FUNCTION_BLOCK POU_MainFunc
VAR_INPUT
END_VAR
VAR_OUTPUT
END_VAR
VAR
	go: BOOL; //local variable to start the program and modes
	TON_0: TON;
	timepass: TIME;
	TimerAmount: TIME:= T#340MS; //this is a specific value type, time of 340ms
	timer2: BOOL;
	Timer1: BOOL;
	TON_1: TON;
	InManual: BOOL;
	Motor: MC_Power;
	onMotor: BOOL;
	Motormove: MC_MoveVelocity;
END_VAR

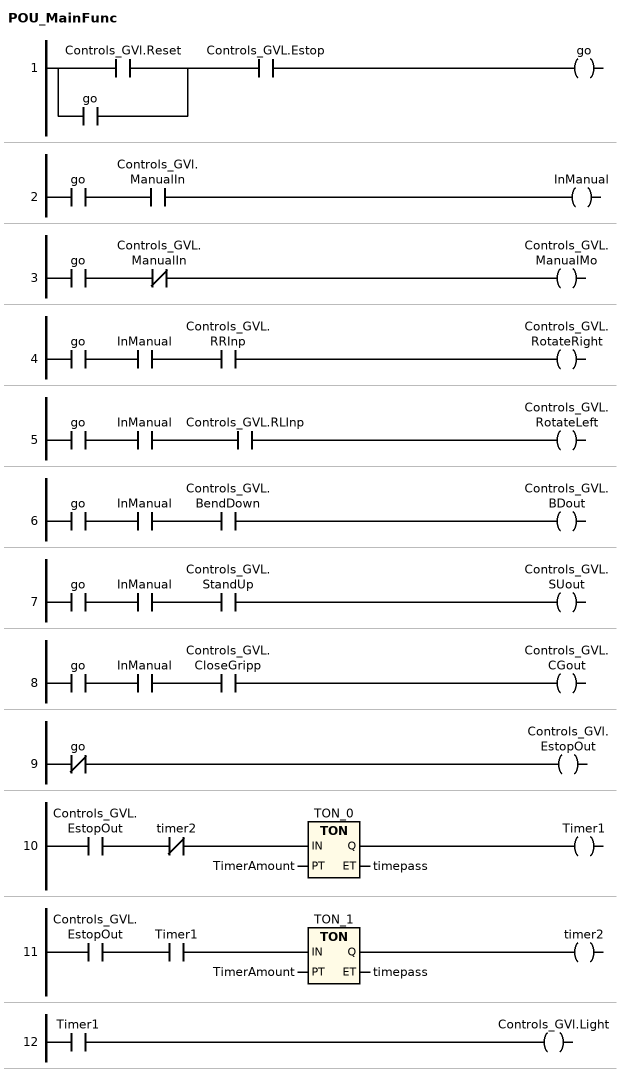
// NETWORK 1
go := (Controls_GVl.Reset OR go) AND Controls_GVL.Estop;

// NETWORK 2
InManual := go AND Controls_GVl.ManualIn;

// NETWORK 3
Controls_GVL.ManualMo := go AND NOT Controls_GVL.ManualIn;

// NETWORK 4
Controls_GVL.RotateRight := go AND InManual AND Controls_GVL.RRInp;

// NETWORK 5
Controls_GVL.RotateLeft := go AND InManual AND Controls_GVL.RLInp;

// NETWORK 6
Controls_GVL.BDout := go AND InManual AND Controls_GVL.BendDown;

// NETWORK 7
Controls_GVL.SUout := go AND InManual AND Controls_GVL.StandUp;

// NETWORK 8
Controls_GVL.CGout := go AND InManual AND Controls_GVL.CloseGripp;

// NETWORK 9
Controls_GVl.EstopOut := NOT go;

// NETWORK 10
TON_0(IN := Controls_GVL.EstopOut AND NOT timer2, PT := TimerAmount, ET => timepass); // TON
Timer1 := TON_0.Q;

// NETWORK 11
TON_1(IN := Controls_GVL.EstopOut AND Timer1, PT := TimerAmount, ET => timepass); // TON
timer2 := TON_1.Q;

// NETWORK 12
Controls_GVl.Light := Timer1;

END_FUNCTION_BLOCK

(* stored: Version 1.1.0.1, ProductVersion 3.1.4024.2
   POU POU_MainFunc: Id {323ec606-e129-471b-a1cc-a5bee963fef0}, SpecialFunc None *)
